// TIA Portal V20 export
VAR_GLOBAL   // PLC tag table "S2_R2"
   S2_R2_Safety1_1 AT %I650.0 : Bool;
   S2_R2_Safety2_1 AT %I650.1 : Bool;
   S2_R2_Safety3_1 AT %I650.2 : Bool;
   S2_R2_Safety4_1 AT %I650.3 : Bool;
   S2_R2_Safety1_2 AT %I650.4 : Bool;
   S2_R2_Safety2_2 AT %I650.5 : Bool;
   S2_R2_Safety3_2 AT %I650.6 : Bool;
   S2_R2_Safety4_2 AT %I650.7 : Bool;
   S2_R2_Valve_Up AT %Q600.0 : Bool;
   S2_R2_Valve_Down AT %Q600.1 : Bool;
   S2_R2_Sen_Drv_1 AT %I600.0 : Bool;
   S2_R2_Sen_Drv_2 AT %I600.1 : Bool;
   S2_R2_Sen_Drv_3 AT %I600.2 : Bool;
   S2_R2_Sen_Drv_4 AT %I600.3 : Bool;
   S2_R2_Sen_Val1_Up AT %I600.4 : Bool;
   S2_R2_Sen_Val1_Down AT %I600.5 : Bool;
   S2_R2_Sen_Val2_Up AT %I600.6 : Bool;
   S2_R2_Sen_Val2_Down AT %I600.7 : Bool;
   S2_R2_Hyd_Filtr AT %I601.0 : Bool;
   S2_R2_Hyd_Empty AT %I601.1 : Bool;
   SS2_R2_ACK_STO AT %Q169.7 : Bool;
   iS2L_Distance_Value AT %IW602 : Int;
   S2_R2_Hydraulic_Unit AT %Q600.2 : Bool;
END_VAR
